// TIA Portal V19 export
DATA_BLOCK "PNIO_Diagnostics_IDB"   // DB18
AUTHOR : NDJH
// stored: InstanceOfName PNIO_Diagnostics, InstanceOfType FB
"PNIO_Diagnostics"
   // VAR
   //    "2_AL1103" { S7_SetPoint := 'True'} : "PNIO_CheckForErrors";
   //    "3_AL1307" { S7_SetPoint := 'True'} : "PNIO_CheckForErrors";
   //    "4_AL1307" { S7_SetPoint := 'True'} : "PNIO_CheckForErrors";
   //    "5_AL1307" { S7_SetPoint := 'True'} : "PNIO_CheckForErrors";
   //    "6_AL1307" { S7_SetPoint := 'True'} : "PNIO_CheckForErrors";
   //    "7_AL1307" { S7_SetPoint := 'True'} : "PNIO_CheckForErrors";
   //    "8_Promag300" { S7_SetPoint := 'True'} : "PNIO_CheckForErrors";
   //    "9_SinaG120" { S7_SetPoint := 'True'} : "PNIO_CheckForErrors";
   //    "10_AL1307" { S7_SetPoint := 'True'} : "PNIO_CheckForErrors";
   //    "11_PNCoup" { S7_SetPoint := 'True'} : "PNIO_CheckForErrors";
   //    "12_AL1307" { S7_SetPoint := 'True'} : "PNIO_CheckForErrors";
   // END_VAR
BEGIN
END_DATA_BLOCK
